Universal Robots PolyScope program: pianobot.urp

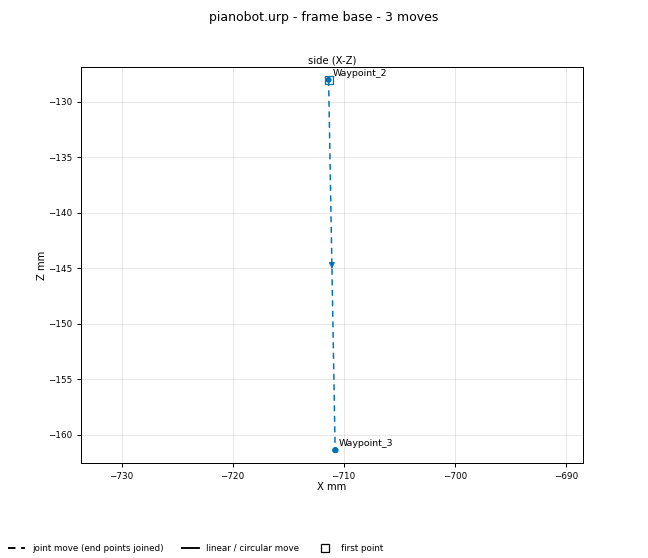
[picture p0: tool path of pianobot.urp in frame base, 3 of 4 moves have a stored position in this frame; points joined in program order, loops and branches not executed]
Program pianobot (installation=default directory=/programs/APS2OsUltimosRomanticos createdIn=3.15.3.106223 lastSavedIn=3.15.3.106223 robotSerialNumber=2017357017)
Calibrated DH parameters: a=[0.0001, -0.032836, -0.39033, 0.000086, 0.000053, 0]; d=[0.089393, 264.548863, -261.578988, -2.85966, 0.094927, 0.082356]; alpha=[1.569373, -0.001603, 0.013671, 1.570599, -1.570158, 0]; deltaTheta=[0.000031, -1.49356, 1.597104, -0.103695, -0.000023, -0.000043]
BeforeStart
  MoveJ speed 60 deg/s, acceleration 80 deg/s^2 (useActiveTCP=false) tcp=TCP_PianoBot
    Waypoint Waypoint_2: TCP in base x=-711.361 y=666.273 z=-128.039 mm, rx=-3.094 ry=0.026 rz=-0.0323 rad; joints [143.259, -170.152, -26.346, -72.891, 87.938, 54.264] deg; flange x=-645.211 y=625.793 z=-28.931 mm, rx=-3.094 ry=0.026 rz=-0.0323 rad
    Waypoint Waypoint_3: TCP in base x=-710.771 y=666.02 z=-161.386 mm, rx=-3.0984 ry=0.0245 rz=-0.043 rad; joints [143.253, -173.368, -24.401, -72.093, 87.916, 54.22] deg; flange x=-645.273 y=626.052 z=-61.64 mm, rx=-3.0984 ry=0.0245 rz=-0.043 rad
  MoveL speed 250 mm/s, acceleration 1200 mm/s^2 (useActiveTCP=true) feature=pianobot
    Waypoint Waypoint_1: TCP in base x=-710.732 y=666.051 z=-161.399 mm, rx=-3.0985 ry=0.0246 rz=-0.0431 rad; joints [143.25, -173.368, -24.4, -72.096, 87.916, 54.223] deg; pose in feature x=0.155 y=0.024 z=0.963 mm, rx=0.0429 ry=0.0104 rz=-0.0001 rad; flange x=-645.24 y=626.08 z=-61.649 mm, rx=-3.0985 ry=0.0246 rz=-0.0431 rad
  Wait Sleep waitTime=5
Robot Program (runOnlyOnce=false)
  Wait Condition expression=start≟1
  escala_mm := p[0.161*escala,0,0,0,0,0]
  var_1 := pose_add(p[0,0,0.001,0.04,0.00,0.0],escala_mm)
  MoveL speed 250 mm/s, acceleration 1200 mm/s^2 (useActiveTCP=false) tcp=TCP_PianoBot; feature=pianobot
    Waypoint Waypoint (Variable): variable=var_1
  Wait Sleep waitTime=0.01
